Staubli VAL3: RosSimpleMsg.pjx

--- RosSimpleMsg.pjx ---
Parameters version=s7.7.2 stackSize=5000 millimeterUnit=true
Program file=start.pgx
Program file=stop.pgx
Data file=RosSimpleMsg.dtx
Type name=Prefix path=Disk://ros_libs/Prefix/Prefix.pjx
Type name=Header path=Disk://ros_libs/Header/Header.pjx

--- RosSimpleMsg.dtx ---
public Header header
  [0]
    num nMsgType
    num nCommType
    num nReplyCode
    num nData[12]
public Prefix prefix
  [0]
    num nLength
    num nData[4]

--- stop.pgx ---
program stop()
begin
end
